(* IEC 61131-3 sources: Elmo_Master/Lasal_PRG/Elmo_EtherCAT_Test_4Axis/Class/TestClass, 1 file *)

(* ---- TestClass.st ---- *)
(*!
<Class
	Name               = "TestClass"
	Revision           = "0.0"
	RealtimeTask       = "false"
	CyclicTask         = "false"
	BackgroundTask     = "false"
	Sigmatek           = "false"
	OSInterface        = "false"
	HighPriority       = "false"
	Automatic          = "false"
	UpdateMode         = "Prescan"
	SharedCommandTable = "true"
	Objectsize         = "(284,120)">
	<Channels>
		<Server Name="ClassSvr" Visualized="false" Initialize="false" WriteProtected="true" Retentive="false"/>
		<Server Name="Server" Visualized="false" Initialize="false" WriteProtected="false" Retentive="false"/>
		<Server Name="Server0" Visualized="false" Initialize="false" WriteProtected="false" Retentive="false"/>
		<Server Name="Server1" Visualized="false" Initialize="false" WriteProtected="false" Retentive="false"/>
		<Server Name="Server2" Visualized="false" Initialize="false" WriteProtected="false" Retentive="false"/>
		<Server Name="Server3" Visualized="false" Initialize="false" WriteProtected="false" Retentive="false"/>
		<Server Name="Server4" Visualized="false" Initialize="false" WriteProtected="false" Retentive="false"/>
		<Server Name="Server5" Visualized="false" Initialize="false" WriteProtected="false" Retentive="false"/>
		<Server Name="Server6" Visualized="false" Initialize="false" WriteProtected="false" Retentive="false"/>
	</Channels>
</Class>
*)
TestClass : CLASS
  //Servers:
	ClassSvr 	: SvrChCmd_DINT;
	Server 	: SvrCh_DINT;
	Server0 	: SvrCh_DINT;
	Server1 	: SvrCh_DINT;
	Server2 	: SvrCh_DINT;
	Server3 	: SvrCh_DINT;
	Server4 	: SvrCh_DINT;
	Server5 	: SvrCh_DINT;
	Server6 	: SvrCh_DINT;
  //Clients:
  //Variables:
  //Functions:
  //Tables:
	FUNCTION @STD
		VAR_OUTPUT
			ret_code	: CONFSTATES;
		END_VAR;
	FUNCTION GLOBAL TAB @CT_;
END_CLASS;
